INTERFACE ITF_Sensor_NO_2InRow_TestDecorator EXTENDS ITF_Sensor_TestDecorator

METHOD PUBLIC SetContact2
VAR_INPUT
	bIN: BOOL;
END_VAR
END_METHOD

END_INTERFACE

(* stored: Version 1.1.0.1
   Itf ITF_Sensor_NO_2InRow_TestDecorator: Id {af78f01e-09ca-42ab-8153-e581f82e560c}
   Method SetContact2: Id {4cf85473-9fa1-43f7-af3e-def32ecc3796} *)
